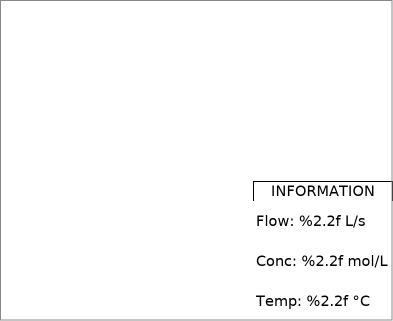
VISUALIZATION WIP  // 393x321
    Group (253,181 140x140)
        Rectangle (0,0 140x140), "INFORMATION"
        Rectangle (0,20 140x40), "Flow: %2.2f L/s", text variable: Flow.out*1000
        Rectangle (0,60 140x40), "Conc: %2.2f mol/L", text variable: Conc.now*1000
        Rectangle (0,100 140x40), "Temp: %2.2f °C", text variable: Temp.now
END_VISUALIZATION

(* stored: Version 1.1.0.1, ProductVersion 3.1.4024.12
   Visu WIP: Id {3864b44c-8849-4f8c-97af-857084cf3c26} *)
